Universal Robots URScript: test.urscript

def test():
movej([-1.494456, -0.482091, -1.710574, -0.709599, 1.032980, 0.368178],a=1,v=0.1)
end
